SUBAPPLICATION Uebung_010f (* AuxFunction2_X1 auf DigitalOutput_Q1 mit GreenWhiteBackground *)
  (* Standard: 61499-2; Description: Copyright (c) 2026 Meisterschulen am Ostbahnhof This program and the accompanying materials are made available under the terms of the Eclipse Public License 2.0 which is available at https://www.eclipse.org/legal/epl-2.0/ SPDX-License-Identifier: EPL-2.0 *)
  (* Version 1.0, 2026-09-06, Franz Höpfinger, Meisterschulen am Ostbahnhof, initial API and implementation and/or initial documentation *)
  PACKAGE Uebungen;
  IMPORT Uebungen::const::UT::DefaultPool::AuxFunction2_X1;
  IMPORT logiBUS::io::DQ::logiBUS_DO::Output_Q1;
  (* Documentation:
  AuxFunction2_X1 auf DigitalOutput_Q1 mit GreenWhiteBackground
   Klassische (nicht-AX-Adapter) Variante von Uebung_010f_AX, aufbauend auf Uebung_010b1: zusätzlich zur Ansteuerung von DigitalOutput_Q1 wird der Zustand von AuxFunction2_X1 als Hintergrundfarbe (grün = EIN, weiß = AUS) zurückgemeldet.
   Funktionsbeschreibung
    - AuxFunction2_X1 (Aux_IX) liefert den booleschen Zustand des zugewiesenen physischen Aux-Tasters/Joysticks über IND/IN.
   - Da klassische EventConnections/DataConnections mehrere Ziele aus einer Quelle erlauben, braucht es - anders als bei der AX-Adapter-Variante - keinen expliziten Split-Baustein: IND und IN gehen direkt sowohl an DigitalOutput_Q1 als auch an GreenWhiteBackground.
   - GreenWhiteBackground2 statt GreenWhiteBackground1, weil AuxFunction2_X1 ein Auxiliary-Function-Type-2-Objekt ist: seine Zuweisung wird sowohl auf dem VT-Bildschirm als auch am Aux-Handle (Joystick) selbst angezeigt. Beide Anzeigen hängen an getrennten Verbindungen und müssen daher separat angesprochen werden (Q_BackgroundColour für das VT, Q_BackgroundColourAux für das Aux-Handle).
    Arbeitsauftrag
   Testen Sie: Aux-Taster drücken/loslassen → Q1 folgt dem Tasterzustand, und die Hintergrundfarbe des Aux-Objekts wechselt gleichzeitig auf dem VT-Bildschirm UND am Aux-Handle selbst zwischen Weiß und Grün.
  *)
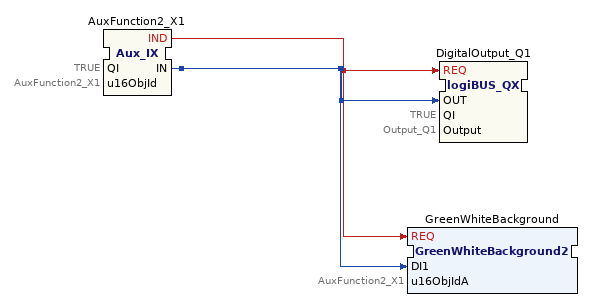
  (* Nachteil: AuxFunction2_X1 muss 2x angegeben werden (Aux_IX.u16ObjId und GreenWhiteBackground.u16ObjIdA). Wichtig: hier MUSS GreenWhiteBackground2 (nicht GreenWhiteBackground1) verwendet werden, weil AuxFunction2_X1 ein Auxiliary-Function-Type-2-Objekt ist - seine Farbe muss sowohl an den VT-Bildschirm als auch an das Aux-Handle (Joystick) selbst gesendet werden. *)
  FBS
    DigitalOutput_Q1 : logiBUS::io::DQ::logiBUS_QX(QI := TRUE, Output := Output_Q1);
    AuxFunction2_X1 : isobus::UT::io::Auxiliary::IN::Aux_IX(QI := TRUE, u16ObjId := AuxFunction2_X1);
  END_FBS
  SUBAPPS
    GreenWhiteBackground : MyLib::sys::GreenWhiteBackground2(u16ObjIdA := AuxFunction2_X1);
  END_SUBAPPS
  EVENT_CONNECTIONS
    AuxFunction2_X1.IND TO DigitalOutput_Q1.REQ;
    AuxFunction2_X1.IND TO GreenWhiteBackground.REQ;
  END_CONNECTIONS
  DATA_CONNECTIONS
    AuxFunction2_X1.IN TO DigitalOutput_Q1.OUT;
    AuxFunction2_X1.IN TO GreenWhiteBackground.DI1;
  END_CONNECTIONS
END_SUBAPPLICATION
